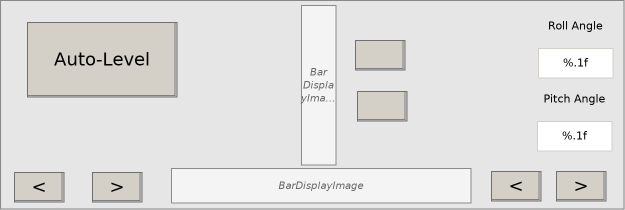
VISUALIZATION ChassisControls  // 625x210
    BarDisplayImage (171,168 300x35), style: BarDisplayImage-Gray, scale format: %.0f, scale -10..10
    BarDisplayImage (301,5 35x160), style: BarDisplayImage-Gray, scale format: %.0f, scale -10..10
    Button (27,22 150x75), "Auto-Level"
    Textfield (538,48 75x30), "%.1f"
    Textfield (537,84 75x30), "Pitch Angle"
    Textfield (538,11 75x30), "Roll Angle"
    Textfield (537,121 75x30), "%.1f"
    Button (14,172 50x30), "<"
    Button (92,172 50x30), ">"
    Button (491,171 50x30), "<"
    Button (556,171 50x30), ">"
    Button (355,40 50x30)
    Button (357,91 50x30)
        p2277200375: -90
END_VISUALIZATION

(* stored: Version 1.1.0.1, ProductVersion 3.1.4024.15
   Visu ChassisControls: Id {ed07c78c-3bc2-4862-b746-deb4f72e80d4} *)
